TYPE CmpWorkStopMainLnSwConfig :
STRUCT
	DBLocation: STRING(30);
END_STRUCT
END_TYPE

(* stored: Version 1.1.0.1, ProductVersion 3.1.4024.6
   DUT CmpWorkStopMainLnSwConfig: Id {c1fa49fa-3872-404a-8dea-73fd2cc0445a} *)
